// TIA Portal V20 export
FUNCTION_BLOCK "FB_SonplasMain"   // FB42, SCL
{ S7_Optimized_Access := 'TRUE' }
// stored: MemoryReserve 100, SetENOAutomatically false
   VAR
      sSonplasLoader : "FB_SonplasLoader";
      iDMC_CodeShuttle1 { S7_SetPoint := 'True'} : String;
      iDMC_CodeShuttle2 : String;
      iDMC_Code : String;
      oDMC_CodeShuttle1 : String;
      oDMC_CodeShuttle2 : String;
      oDMC_Code : String;
   END_VAR
   VAR_TEMP
      tRetMov : Int;
      tIndex : Int;
   END_VAR
BEGIN
   REGION Description head
       //==================================================================================
       // POSALUX Swiss SA / (C) Copyright 2025
       //----------------------------------------------------------------------------------
       // Title: Digital Inputs mapping
       // Comment/Function: Digital Inputs mapping
       // Author: Fabien WALDT
       // Engineering: TIA Portal v17
       //----------------------------------------------------------------------------------
       // Change log table:
       // Version  | Date     | Expert in charge | Changes applied
       // ---------|----------|------------------|-----------------------------------------
       // 00.00.01 | 20250423 | WFA              | First released version
       // =================================================================================
   END_REGION

   REGION DMC Reading
      // Transfer DMC Code Shuttle 1 (IB204-IB223)
       // #tRetMov := MOVE_BLK_VARIANT(SRC := P# I204.0 BYTE 20, // WAF COMENTAIRE POUR TESTS TRACABILITE
       //                              COUNT := 20,
       //                              SRC_INDEX := 0,
       //                              DEST_INDEX := 0,
       //                              DEST => #sSonplasLoader.iPartInDMC_CodeShuttle1);

       // String Conversion
       #iDMC_CodeShuttle1 := '';
       FOR #tIndex := 0 TO 19 DO
           IF #sSonplasLoader.iPartInDMC_CodeShuttle1[#tIndex] <> 0 THEN
               #iDMC_CodeShuttle1 := CONCAT(IN1 := #iDMC_CodeShuttle1, IN2 := CHAR_TO_STRING(BYTE_TO_CHAR(#sSonplasLoader.iPartInDMC_CodeShuttle1[#tIndex])));
           END_IF;
       END_FOR;

      // Transfer DMC Code Shuttle 2 (IB224-IB243)
       // #tRetMov := MOVE_BLK_VARIANT(SRC := P# I224.0 BYTE 20, // WAF COMENTAIRE POUR TESTS TRACABILITE
       //                             COUNT := 20,
       //                             SRC_INDEX := 0,
       //                             DEST_INDEX := 0,
       //                             DEST => #sSonplasLoader.iPartInDMC_CodeShuttle2);


       // String Conversion
      #iDMC_CodeShuttle2 := '';
       FOR #tIndex := 0 TO 19 DO
           IF #sSonplasLoader.iPartInDMC_CodeShuttle2[#tIndex] <> 0 THEN
               #iDMC_CodeShuttle2 := CONCAT(IN1 := #iDMC_CodeShuttle2, IN2 := CHAR_TO_STRING(BYTE_TO_CHAR(#sSonplasLoader.iPartInDMC_CodeShuttle2[#tIndex])));
           END_IF;
       END_FOR;

       // Transfer DMC Code (IB247-IB266)
       #tRetMov := MOVE_BLK_VARIANT(SRC := P# I247.0 BYTE 20,
                                    COUNT := 20,
                                    SRC_INDEX := 0,
                                    DEST_INDEX := 0,
                                    DEST => #sSonplasLoader."iPartInDMC Code");


       // String Conversion
       #iDMC_Code := '';
       FOR #tIndex := 0 TO 19 DO
           IF #sSonplasLoader."iPartInDMC Code"[#tIndex] <> 0 THEN
               #iDMC_Code := CONCAT(IN1 := #iDMC_Code, IN2 := CHAR_TO_STRING(BYTE_TO_CHAR(#sSonplasLoader."iPartInDMC Code"[#tIndex])));
           END_IF;
       END_FOR;

   END_REGION

   REGION Sonplas Loader
       #sSonplasLoader(iOperateInDiagDPCoupler:="DB_DigitalInputsSonplas".sSonplasDiagDPCoupler.sSWStatus,
                       iOperateInReady:="DB_DigitalInputsSonplas".sSonplasReady.sSWStatus,
                       iOperateInNoEStop:="DB_DigitalInputsSonplas".sSonplasNoEStop.sSWStatus,
                       iOperateInDoorsClosed:="DB_DigitalInputsSonplas".sSonplasDoorsClosed.sSWStatus,
                       iOperateInRunError:="DB_DigitalInputsSonplas".sSonplasRunError.sSWStatus,
                       iOperateInOutCollision:="DB_DigitalInputsSonplas".sSonplasOutCollision.sSWStatus OR "DB_WAF".Sonplas.OperateInOutCollision,
                       iPartInShuttle1Finished:="DB_DigitalInputsSonplas".sSonplasShuttle1Finished.sSWStatus,
                       iPartInShuttle2Finished:="DB_DigitalInputsSonplas".sSonplasShuttle2Finished.sSWStatus,
                       iMeasureInFlowResultAvail:="DB_DigitalInputsSonplas".sSonplasFlowResultAvail.sSWStatus,
                       iMeasureInFlowResult:= WORD_TO_INT(SWAP_WORD("AI_SonplasFlowResult")),
                       oOperateOutDiagDPCoupler=>"DB_DigitalOutputs".sSonplasDiagDPCoupler.sSWStatus,
                       oOperateOutReady=>"DB_DigitalOutputs".sSonplasReady.sSWStatus,
                       oOperateOutNoEStop=>"DB_DigitalOutputs".sSonplasNoEStop.sSWStatus,
                       oOperateOutDoorsClosed=>"DB_DigitalOutputs".sSonplasDoorsClosed.sSWStatus,
                       oOperateOutRunError=>"DB_DigitalOutputs".sSonplasRunError.sSWStatus,
                       oPartOutShuttle1InPos=>"DB_DigitalOutputs".sSonplasShuttle1InPos.sSWStatus,
                       oPartOutPart1OK=>"DB_DigitalOutputs".sSonplasPart1OK.sSWStatus,
                       oPartOutPart1NOK=>"DB_DigitalOutputs".sSonplasPart1NOK.sSWStatus,
                       oPartOutShuttle2InPos=>"DB_DigitalOutputs".sSonplasShuttle2InPos.sSWStatus,
                       oPartOutPart2OK=>"DB_DigitalOutputs".sSonplasPart2OK.sSWStatus,
                       oPartOutPart2NOK=>"DB_DigitalOutputs".sSonplasPart2NOK.sSWStatus,
                       oMeasureOutResultAccepted=>"DB_DigitalOutputsSonplas".Sonplas_ResultAccepted.sSWStatus);
   END_REGION

   REGION DMC Writing   
       // Transfer DMC Code Shuttle 1 (QB204-QB223)
       FOR #tIndex := 1 TO LEN(#oDMC_CodeShuttle1) DO
           #sSonplasLoader.oPartOutDMC_CodeShuttle1[#tIndex - 1] := CHAR_TO_BYTE(#oDMC_CodeShuttle1[#tIndex]);
       END_FOR;

       #tRetMov := MOVE_BLK_VARIANT(SRC := #sSonplasLoader.oPartOutDMC_CodeShuttle1,
                                    COUNT := 20,
                                    SRC_INDEX := 0,
                                    DEST_INDEX := 0,
                                    DEST => P# Q204.0 BYTE 20);

   // Transfer DMC Code Shuttle 2 (QB224-QB243)
   FOR #tIndex := 1 TO LEN(#oDMC_CodeShuttle2) DO
       #sSonplasLoader.oPartOutDMC_CodeShuttle2[#tIndex - 1] := CHAR_TO_BYTE(#oDMC_CodeShuttle2[#tIndex]);
   END_FOR;

   #tRetMov := MOVE_BLK_VARIANT(SRC := #sSonplasLoader.oPartOutDMC_CodeShuttle2,
                                COUNT := 20,
                                SRC_INDEX := 0,
                                DEST_INDEX := 0,
                                DEST => P# Q224.0 BYTE 20);

   // Transfer DMC Code (QB247-QB266)
   FOR #tIndex := 1 TO LEN(#oDMC_Code) DO
       #sSonplasLoader.oPartOutDMC_Code[#tIndex - 1] := CHAR_TO_BYTE(#oDMC_Code[#tIndex]);
   END_FOR;

   #tRetMov := MOVE_BLK_VARIANT(SRC := #sSonplasLoader.oPartOutDMC_Code,
                                COUNT := 20,
                                SRC_INDEX := 0,
                                DEST_INDEX := 0,
                                DEST => P# Q247.0 BYTE 20);
   END_REGION
END_FUNCTION_BLOCK
